FUNCTION_BLOCK Q_SelectActiveWorkingSet (* Command Hide/Show Object (Container) ( Part 6 - F.2 ) *)
  (* Standard: ISO 11783-6; Description: Command Select Active Working Set( Part 6 - F.64 ) Return values iso_s16 - E_NO_ERR - OK - E_OVERFLOW - buffer overflow - E_NOACT - Command not possible in current state - E_NO_INSTANCE - No VT client available *)
  (* Version 1.0, 2022-07-08, franz *)
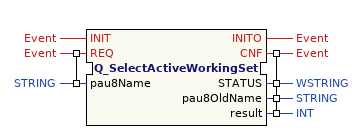
  EVENT_INPUT
    INIT; (* Service Initialization *)
    REQ WITH pau8Name; (* Service Request *)
  END_EVENT
  EVENT_OUTPUT
    INITO; (* Initialization Confirm *)
    CNF WITH STATUS, pau8OldName, result; (* Confirmation of Requested Service *)
  END_EVENT
  VAR_INPUT
    pau8Name : STRING; (* Iso NAME of the new active working set *)
  END_VAR
  VAR_OUTPUT
    STATUS : WSTRING; (* Service Status *)
    pau8OldName : STRING; (* Old value of Visible *)
    result : INT; (* retval see description *)
  END_VAR
END_FUNCTION_BLOCK
